FUNCTION_BLOCK Delay
VAR_INPUT
END_VAR
VAR_OUTPUT
END_VAR
VAR
	
	delay : TON;
    Count : INT := 0;

	
END_VAR

Delay(IN:=TRUE, PT:=T#5S);
IF NOT(Delay.Q) THEN
   RETURN;
END_IF
Delay(IN:=FALSE);

END_FUNCTION_BLOCK

(* stored: Version 1.1.0.1, ProductVersion 3.1.4024.15
   POU Delay: Id {f44b84ec-03f4-489c-8e59-7254caf2a04b}, SpecialFunc None *)
